FUNCTION_BLOCK FB_ABL_110_Feeder
(****************************************************************************************)
(*	TITEL				RFID-Ring laden, Feeder and rotary table                        *)
(*	Status				ungetestet                         								*)
(*	Beschrieb:			Ablaufbeschreibung												*)
(*																						*)
(*	Steps:	self-explained using enum													*)
(***********************************Revisionen*******************************************)
(*	see github blames																	*)
(****************************************************************************************)

VAR_INPUT
    xIN_Reset       : BOOL;          // Schrittkette zurücksetzen 
    xIN_Init        : BOOL;          // Initialisieren
    xIN_Quit        : BOOL;          // Fehler quittieren 
    xIN_Start       : BOOL;          // Startbefehl
    xIN_Sperre      : BOOL;          // FB Sperren 
    xIN_NextStep    : BOOL;          // Nächsten Schritt ausführen 
    xIN_AlarmAktiv  : BOOL;          // Anlage hat Alarm
    xIN_DryCycle    : BOOL;          // Fahren ohne Teile
    xIN_RestartCYCL : BOOL;          // Zyklus erneut starten im STEP, END, LEERFAHREN
    enIN_State      : enState;       // Status Anlage
    tIN_Timeout     : TIME := T#10s; // Timout

    pxFG_Freigabe : POINTER TO BOOL; //Freigabe von Station

    // Application specific
    xIN_PickPiece : BOOL; (* signal from the pick and place element
                             the number of picked signal depend on the recipe *)
    xIN_RotTableBlockedByPnp : BOOL; // Is the pick and place blocking the rotary table?
END_VAR
VAR_OUTPUT
    (* standart Ausgänge *)
    xOUT_ErrFlag  : BOOL;           // Error Flag 
    xOUT_Busy     : BOOL;           // Baustein befindet sich im Ablauf 
    xOUT_Done     : BOOL;           // Baustein hat den Ablauf beendet 		
    xOUT_Ready    : BOOL;           // Ready to begin, should be the same state as done	
    xOUT_Timeout  : BOOL;           // Timeout FB 
    xOUT_InitDone : BOOL;           // initialisierung fertig
    xOUT_Wait     : BOOL;           // Wartet auf Bedingung
    iOUT_Step     : ST110_Feeder_e; // Aktueller Schritt 
    sOUT_Step     : STRING;         // Aktueller Schritt but in string format
    bOUT_Error    : BYTE;           // Fehlernummer

    // Application specific
    xOUT_PceReadyToPick : BOOL; // the piece(s) is/are ready to picked
END_VAR
VAR
    (* Standard *)
    (* Schritt *)
    iLastStep : ST110_Feeder_e; // Merker letzter Schritt 
    iPreStep  : ST110_Feeder_e; // Schritt zurück nach Alarm 
    iAktStep  : ST110_Feeder_e; // aktueller Schritt

    // Trigger Starten 
    rtSTART : R_TRIG;
    // Timer TimeOut 
    TON_Timeout : TON;

    (* Bausteine *)
	btfb_feeder					: FB_BUTTON;

    // Application specific
    fb_axis110_10W               : FB_AxisLMturn_V1_1;
    simu_axis110_10W             : FB_Simu_AxisLM_V1_1;
    fb_feeder                    : FB_Feeder2Sensors;
    fifo                         : FB_Fifo(3);
    simu_feeder                  : FB_Simu_Feeder; // simulation of a feeder
    simu_fifo_feeder_to_rotTable : FB_Fifo(20);    // fifo to hold a piece
    rtPutPiece                   : R_TRIG;         // trigger to add a piece

    rtPick : R_TRIG; // r_trig signal from the pick and place machine

    iCurrentTableIndex : INT; // current table index
    iSearchIndex       : INT; (* Initialization index TO see how many element we have AT startup
                                 or after an alarm *)

    ton_wait_blow_piece : TON;
    tof_color_sensor    : TOF;

	rTest : REAL;
END_VAR
VAR CONSTANT
    MAX_SEARCH_TURN : INT := 3; // maximum search number

    FEEDER_SIMULATION : BOOL := TRUE; // Simulate this code
END_VAR

(*******************************************************************)
(* Trigger  *)
(*******************************************************************)
(* Zurücksetzen *)
IF xIN_RESET THEN
    iPreStep  := ST110_Feeder_e.RESET;
    iOUT_Step := ST110_Feeder_e.RESET;
END_IF;

(* Error Quittieren *)
IF (bOUT_Error <> 0) AND xIN_Quit THEN
    xOUT_ErrFlag := FALSE;
    bOUT_Error   := 0;
    iOUT_Step    := iPreStep;
END_IF;

iCurrentTableIndex := iCurrentTableIndex MOD 3;

(*******************************************************************)
(* Timer *)
(*******************************************************************)
TON_Timeout(IN := xIN_NextStep AND (iLastStep = iOUT_Step) (*todo FG *) ,
            PT := tIN_Timeout);

// we use a set reset to be sure that the blower blow event if the time
// is not elapsed
IF IO_BOX.I8004_ST110_farbsensor_lagekontrolle THEN
    ton_wait_blow_piece.IN := TRUE;

ELSIF NOT IO_BOX.I8004_ST110_farbsensor_lagekontrolle AND ton_wait_blow_piece.Q THEN
    ton_wait_blow_piece.IN := FALSE;

END_IF

ton_wait_blow_piece(IN :=, // see code above
                    PT := DINT_TO_TIME(_20_AUTO.recipe.st110.waitBlowPieceTon_ms));

tof_color_sensor(IN := ton_wait_blow_piece.Q,
                 PT := DINT_TO_TIME(_20_AUTO.recipe.st110.blowPieceTof_ms));

(*******************************************************************)
(* Bausteine *)
(*******************************************************************)
btfb_feeder(pbtIN  := ADR(HMI.btManuCylinders[StationList_e.ST110][3]),
            xINdis := (enIN_State <> enState.StateMANU),
            xINon  :=,
            xINerr := fb_feeder.xOUT_Empty);

IF btfb_feeder.pbtIN^.rtrig THEN
    btfb_feeder.xINon := NOT btfb_feeder.xINon;
ELSIF (enIN_State <> enState.StateMANU) THEN
    btfb_feeder.xINon := FALSE;
END_IF;

fb_feeder(xIN_Enable := ((enIN_State <= enState.StateAUTO) AND (enIN_State >= enState.StateSTEP)) OR btfb_feeder.xINon,
          xIN_PieceInEnd
              := TRUE, // IO_BOX.I6000_ST110_teil_in_vereinzelung, 
          xIN_PieceMax              := IO_BOX.I8001_ST110_maximum,
          xIN_InSimulation          := FEEDER_SIMULATION AND CONST.USE_SIMULATION,
          refIN_SimulatedFifo       := simu_fifo_feeder_to_rotTable,
          iIN_FifoSetMaxSensorValue := 10,
          diIN_SignlFilter_ms       := _20_AUTO.recipe.st110.FeederConfig.InFilterDelay,
          diIN_StartDelay_ms        := _20_AUTO.recipe.st110.FeederConfig.StartDelay,
          diIN_StopDelay_ms         := _20_AUTO.recipe.st110.FeederConfig.StopDelay,
          diIN_EmptyDelay_ms        := _20_AUTO.recipe.st110.FeederConfig.EmptyDelay);

simu_feeder(xIN_Enable         := fb_feeder.xOUT_EnableFeeder AND FEEDER_SIMULATION AND CONST.USE_SIMULATION,
            xIN_PceSensor      := fb_feeder.xIN_PieceInEnd,
            tIN_NewPieceTime   := 500,
            iIN_WaitTimeMin_ms := 500,
            iIN_WaitTimeMax_ms := 1000);

rtPick(CLK := xIN_PickPiece);
rtPutPiece(CLK := simu_feeder.xOUT_NewPiece);

IF rtPutPiece.Q AND NOT simu_fifo_feeder_to_rotTable.IsFull() THEN
    simu_fifo_feeder_to_rotTable.Put(1);
END_IF

IF ST110_Feeder_e.Init_simu_home_table = iOUT_Step THEN
    fb_axis110_10W.rIN_Position := TO_REAL(120.0 - LMOD(ST110_Axis.axis110_10W.rActPos, 120.0));

ELSE
    fb_axis110_10W.rIN_Position := 120.0;

END_IF

simu_axis110_10W(xIN_Enable          := FEEDER_SIMULATION AND CONST.USE_SIMULATION,
                 wIN_AxisState       := ST110_Axis.axis110_10W.wState,
                 bIN_AxisCntr        := fb_axis110_10W.bOUT_AxisCntr,
                 udiIN_HomingTime_ms := 1000,
                 pIN_axisSimu        := ADR(SIMU.axis_ref[Axis_e.ST110_10W]),
                 pIN_axisHW          := ADR(ST110_Axis.axis110_10W.axis),
                 rIN_PosActual       := fb_axis110_10W.rOUT_ActPos,
                 rIN_PosMax          := ST110_Axis.const110_10W.POS_MAX,
                 rIN_PosMin          := ST110_Axis.const110_10W.POS_MIN,
                 rIN_PixMax          := 0,
                 rIN_PixMin          := 0);

fb_axis110_10W(enIN_State     := enIN_State,
               parIN_Buttons  := ADR(AXIS.btTeachArAxis[Axis_e.ST110_10W]),
               xIN_DisButtons :=,
               xIN_Quit       := xIN_Quit,
               xIN_PARAMok    := TRUE,
               xIN_FREE       := NOT xIN_RotTableBlockedByPnp,
               xIN_FREE_HOME  := TRUE,
               rIN_POSMIN     := ST110_Axis.const110_10W.POS_MIN,
               rIN_POSMAX     := ST110_Axis.const110_10W.POS_MAX,
               rIN_VELOMAX    := ST110_Axis.const110_10W.VELO_MAX,
               rIN_VELOMANU   := ST110_Axis.const110_10W.VELO_MANU,
               rIN_VELOOPEN   := ST110_Axis.const110_10W.VELO_MANU / 4,
               rIN_JogInc     := AXIS.rTeachIncAxis,
               xIN_Execute    := ST110_Feeder_e.Init_set_table_pos = iOUT_Step OR
                                 ST110_Feeder_e.Init_table_go_to_zero = iOUT_Step OR
                                 ST110_Feeder_e.Init_simu_home_table = iOUT_Step OR
                                 ST110_Feeder_e.load_piece = iOUT_Step OR
                                 ST110_Feeder_e.wait_rotary_table_done = iOUT_Step,
               xIN_Relative     := fb_axis110_10W.xIN_Execute,
               xIN_STOP         := FALSE,
               xIN_OFF          := FALSE,
               rIN_Position     :=, // Is set above
               rIN_Velocity     := TO_REAL(100.0),
               rIN_Acceleration := TO_REAL(1440.0),
               rIN_Deceleration := TO_REAL(1440.0),
               rIN_Jerk         := TO_REAL(720000.0),
               xIN_Home         := ST110_feeder_e.Init_home_table = iOUT_Step,
               xIN_Reset        := xIN_Reset OR ST110_feeder_e.RESET = iOUT_Step,
               // The simu fb gives us the hardware signal when we are not in simulation
               wAxisState    := simu_axis110_10W.wOUT_AxisState,
               bOUT_AxisCntr => ST110_Axis.axis110_10W.bCtrlHi,
               rOUT_ActPos   =>, // leave empty, rActPos must be set using the modulo
               axisIN_REF    := simu_axis110_10W.pOUT_axisRef^);

ST110_Axis.axis110_10W.rActPos := LREAL_TO_REAL(simu_axis110_10W.pOUT_axisRef^.NcToPlc.ModuloActPos);

(*******************************************************************)
(* OUTPUTS *)
(*******************************************************************)
// Error Flag 
xOUT_ErrFlag := (bOUT_Error <> 0) OR (ST110_Feeder_e.ERROR = iOUT_Step);
// Baustein befindet sich im Ablauf 
xOUT_Busy := (iOUT_Step > ST110_Feeder_e.READY) AND (iOUT_Step < ST110_Feeder_e.DONE);
// Baustein hat den Ablauf beendet
xOUT_Done := (iOUT_Step = ST110_Feeder_e.DONE);
// Process ready
xOUT_Ready := (iOUT_Step = ST110_Feeder_e.READY);
// Timeout FB 				 		
xOUT_Timeout := TON_Timeout.Q;
// Itialisierung fertig			
xOUT_InitDone := (iOUT_Step = ST110_Feeder_e.READY);
// Aktueller Schritt			
iOUT_Step := iOUT_Step; //Im Ablauf gesetzt		
sOUT_Step := TO_STRING(iOUT_Step);
//Fehlernummer	 
bOUT_Error := bOUT_Error; //Im Ablauf/FB gesetzt	
(* Warte (alle Schritte wo auf FG oder Teile gewartet wird) *)
xOUT_Wait := (iOUT_Step = ST110_Feeder_e.DONE);

// TODO add simulation constant to prevent the output to be set
IO_BOX.Q8000_ST110_freigabe_wf    := fb_feeder.xOUT_EnableFeeder AND NOT (FEEDER_SIMULATION AND CONST.USE_SIMULATION);
IO_BOX.Q8003_ST110_forderband_ein :=
    (enIN_State >= enState.StateLEER) AND
    NOT (FEEDER_SIMULATION AND CONST.USE_SIMULATION);

// blow out

IO_BOX.Q8005_ST110_blow_piece := fb_feeder.xOUT_EnableFeeder AND
                                 tof_color_sensor.Q AND
                                 NOT (FEEDER_SIMULATION AND CONST.USE_SIMULATION);

(*******************************************************************)
(* Ablauf *)
(*******************************************************************)

(* Sperren *)
IF xIN_Sperre THEN
    iPreStep  := ST110_Feeder_e.RESET;
    iOUT_Step := ST110_Feeder_e.RESET;
    RETURN;
END_IF;

(* Schritt Merker *)
IF iAktStep <> iOUT_Step THEN
    iLastStep := iAktStep;
    iAktStep  := iOUT_Step;
END_IF

(* START *)
rtSTART(CLK := xIN_Start);

IF 0 = bOUT_Error THEN
    IF fb_axis110_10W.xOUT_ErrFlag THEN
        bOUT_Error := 11;
    END_IF
ELSIF iOUT_Step < ST110_Feeder_e.ERROR THEN
    iOUT_Step := ST110_Feeder_e.ERROR;
END_IF

(*******************************************************************)
(* Schrittkette  *)
(*******************************************************************)
CASE iOUT_Step OF

(***** RESET *****)
ST110_Feeder_e.RESET: (* Schritt 0-99 *)
    //Initialisierungen
    //Start Init Ablauf
    IF xIN_Init THEN
        iOUT_Step := ST110_Feeder_e.INIT;
        //Start Manu Ablauf
    ELSIF enIN_State = StateMANU AND xIN_NextStep THEN
        iOUT_Step := ST110_Feeder_e.INIT;
    END_IF;

(***** INIT *****)
ST110_Feeder_e.INIT: (* Grundstellung ? *)
    IF NOT xIN_RotTableBlockedByPnp THEN
        iOUT_Step := ST110_Feeder_e.Init_home_table;
    END_IF

ST110_Feeder_e.Init_home_table:
    IF fb_axis110_10W.xOUT_HOMED THEN
        iCurrentTableIndex := 0;

        IF FEEDER_SIMULATION AND CONST.USE_SIMULATION THEN
            iOUT_Step := ST110_Feeder_e.Init_simu_home_table;
        ELSE
            iOUT_Step := ST110_Feeder_e.Init_reset_search_index;
        END_IF
    END_IF

ST110_Feeder_e.Init_simu_home_table:
    IF fb_axis110_10W.xOUT_DONE THEN
        iOUT_Step := ST110_Feeder_e.Init_reset_search_index;
    END_IF

ST110_Feeder_e.Init_table_go_to_zero:
    IF fb_axis110_10W.xOUT_DONE THEN
        iOUT_Step := ST110_Feeder_e.Init_reset_search_index;
    END_IF

ST110_Feeder_e.Init_reset_search_index:
    iSearchIndex := 0;
    fifo.Empty();
    iOUT_Step := ST110_Feeder_e.READY; // Bypass search algorithm, unusful

ST110_Feeder_e.Init_set_table_pos:
    IF fb_axis110_10W.xOUT_DONE THEN
        iCurrentTableIndex := iCurrentTableIndex + 1;
        iOUT_Step          := ST110_Feeder_e.Init_see_if_piece_there;
    END_IF

ST110_Feeder_e.Init_see_if_piece_there:
    IF simu_feeder.xOUT_NewPiece THEN
        fifo.Put(1);
    END_IF

    IF iSearchIndex < MAX_SEARCH_TURN THEN
        iOUT_Step    := ST110_Feeder_e.Init_set_table_pos;
        iSearchIndex := iSearchIndex + 1;
    ELSE
        iOUT_Step := ST110_Feeder_e.READY;
    END_IF

(***** READY / INIT DONE *****)
ST110_Feeder_e.READY: (* Start AUTO,END,LEER,STEP *)
    IF xIN_Start THEN //IF rtSTART.Q THEN
        iOUT_Step := ST110_Feeder_e.START;
    END_IF

(***** START  ZYKLISCH *****)
ST110_Feeder_e.START: (*  *)
    IF xIN_NextStep AND pxFG_Freigabe^ THEN
        iOUT_Step := ST110_Feeder_e.check_if_feeding_necessary;
    END_IF;

ST110_Feeder_e.check_if_feeding_necessary:
    IF fifo.IsFull() THEN
        iOUT_Step := ST110_Feeder_e.DONE;
    ELSE
        iOUT_Step := ST110_Feeder_e.wait_on_a_piece;
    END_IF

ST110_Feeder_e.wait_on_a_piece:
    IF (FEEDER_SIMULATION AND CONST.USE_SIMULATION AND NOT simu_fifo_feeder_to_rotTable.IsEmpty()) OR
       (NOT (FEEDER_SIMULATION AND CONST.USE_SIMULATION) AND IO_BOX.I6000_ST110_teil_in_vereinzelung) THEN
        iOUT_Step := ST110_Feeder_e.load_piece;
        simu_fifo_feeder_to_rotTable.Pop(1);
    END_IF

ST110_Feeder_e.load_piece:
    IF NOT fb_axis110_10W.xOUT_DONE THEN
        iOUT_Step := ST110_Feeder_e.wait_rotary_table_done;
    END_IF

ST110_Feeder_e.wait_rotary_table_done:
    IF fb_axis110_10W.xOUT_DONE THEN
        fifo.Put(1);
        iOUT_Step := ST110_Feeder_e.check_if_feeding_necessary;
    END_IF

(***** DONE *****)
ST110_Feeder_e.DONE: (* Letzter Schritt  *)
    IF rtPick.Q THEN
        fifo.Pop(TO_INT(_20_AUTO.recipe.st110.xUseVerLeft));
        fifo.Pop(TO_INT(_20_AUTO.recipe.st110.xUseVerRight));
    END_IF

    IF NOT xIN_AlarmAktiv THEN
        //AUTO
        IF (enIN_State = StateAUTO) AND xIN_RestartCYCL AND NOT fifo.IsFull() THEN
            iOUT_Step := ST110_Feeder_e.START;
            //STEP / END / LEERFAHREN restart
        ELSIF (enIN_State < StateAUTO) AND (enIN_State >= enState.StateSTEP) AND xIN_RestartCYCL AND NOT fifo.IsFull()
            THEN
            iOUT_Step := ST110_Feeder_e.START;
            //STEP / END / LEERFAHREN fertig
        ELSIF (enIN_State = StateREADY) THEN
            iOUT_Step := ST110_Feeder_e.READY;
        END_IF;
    END_IF;

(************ ERROR *************)
ST110_Feeder_e.ERROR: (* ERROR *) ;

END_CASE;

END_FUNCTION_BLOCK

(* stored: Version 1.1.0.1, ProductVersion 3.1.4024.6
   POU FB_ABL_110_Feeder: Id {939c70cc-58c9-4d34-aa7b-700c761a72fe}, SpecialFunc None *)
